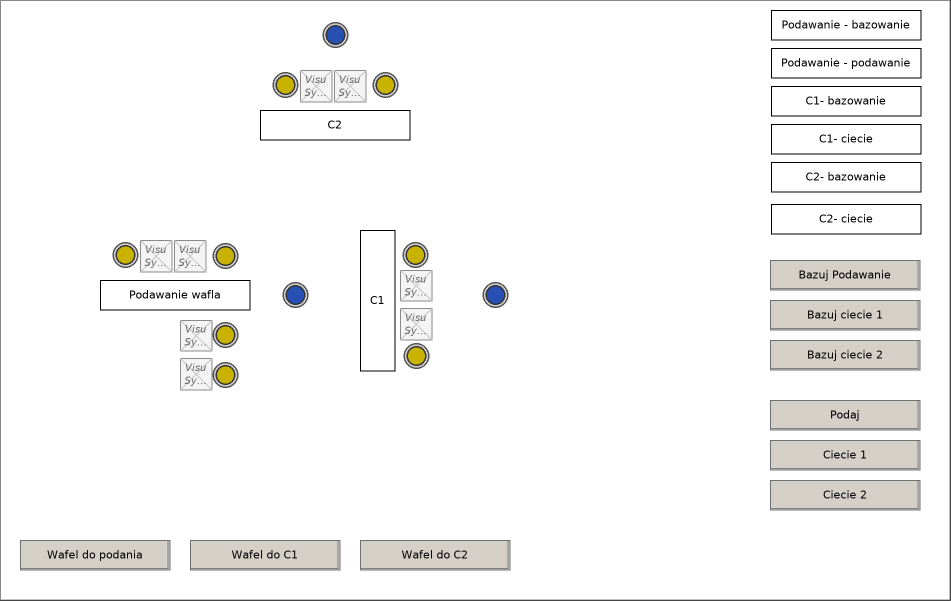
VISUALIZATION Symulacja  // 951x601
VAR_IN_OUT
	stDane									: DUT_Wizualizacja_SymulacjaDane;
END_VAR
    Line (950,0) (950,600)
    Line (0,600) (950,600)
    Rectangle (100,280 150x30), "Podawanie wafla"
    Rectangle (360,230 35x141), "C1"
    Rectangle (260,110 150x30), "C2"
    Lamp1 (401,341 31x30), variable: stDane.bCiecie1_Poczatek, style: Lamp-Lamp1-Yellow
    Lamp1 (400,240 31x30), variable: stDane.bCiecie1_Koniec, style: Lamp-Lamp1-Yellow
    Lamp1 (270,70 31x30), variable: stDane.bCiecie2_Poczatek, style: Lamp-Lamp1-Yellow
    Lamp1 (370,70 31x30), variable: stDane.bCiecie2_Koniec, style: Lamp-Lamp1-Yellow
    Lamp1 (110,240 31x30), variable: stDane.bPodawaniePrzesuwanieKoniec, style: Lamp-Lamp1-Yellow
    Lamp1 (210,241 31x30), variable: stDane.bPodawaniePrzesuwaniePoczatek, style: Lamp-Lamp1-Yellow
    Lamp1 (210,320 31x30), variable: stDane.bPodawanieZabierakKoniec, style: Lamp-Lamp1-Yellow
    Lamp1 (210,360 31x30), variable: stDane.bPodawanieZabierakPoczatek, style: Lamp-Lamp1-Yellow
    Lamp1 (280,280 31x30), variable: stDane.bCzujnikWaflaDoPodania, style: Lamp-Lamp1-Blue
    Lamp1 (480,280 31x30), variable: stDane.bCzujnikWaflaDoCiecia1, style: Lamp-Lamp1-Blue
    Lamp1 (320,20 31x30), variable: stDane.bCzujnikWaflaDoCiecia2, style: Lamp-Lamp1-Blue
    Rectangle (771,10 150x30), "Podawanie - bazowanie", colour toggle: stDane.stStanySilownikow.bPodawanie_Bazowanie
    Rectangle (771,48 150x30), "Podawanie - podawanie", colour toggle: stDane.stStanySilownikow.bPodawanie_Podawanie
    Rectangle (771,86 150x30), "C1- bazowanie", colour toggle: stDane.stStanySilownikow.bCiecie1_Bazowanie
    Rectangle (771,124 150x30), "C1- ciecie", colour toggle: stDane.stStanySilownikow.bCiecie1_Ciecie
    Rectangle (771,162 150x30), "C2- bazowanie", colour toggle: stDane.stStanySilownikow.bCiecie2_Bazowanie
    Rectangle (771,204 150x30), "C2- ciecie", colour toggle: stDane.stStanySilownikow.bCiecie2_Ciecie
    Image (180,358 32x32), invisible if: Not stDane.stStanySilownikow.bPodawanie_Zabierak_WStronePoczatku, image: VisuSymbols.Symbols.ArrowBoldDown
    Image (180,320 32x31), invisible if: Not stDane.stStanySilownikow.bPodawanie_zabierak_WStroneKonca, image: VisuSymbols.Symbols.ArrowBoldUp
    Image (140,240 32x32), invisible if: Not stDane.stStanySilownikow.bPodawanie_Przesuwanie_WStroneKonca, image: VisuSymbols.Symbols.ArrowBoldLeft
    Image (174,240 32x32), invisible if: Not stDane.stStanySilownikow.bPodawanie_Przesuwanie_WStronePoczatku, image: VisuSymbols.Symbols.ArrowBoldRight
    Image (400,308 32x32), invisible if: Not stDane.stStanySilownikow.bCiecie1_Naped_WStronePoczatku, image: VisuSymbols.Symbols.ArrowBoldDown
    Image (400,270 32x31), invisible if: Not stDane.stStanySilownikow.bCiecie1_Naped_WStroneKonca, image: VisuSymbols.Symbols.ArrowBoldUp
    Image (300,70 32x32), invisible if: Not stDane.stStanySilownikow.bCiecie2_Naped_WStronePoczatku, image: VisuSymbols.Symbols.ArrowBoldLeft
    Image (334,70 32x32), invisible if: Not stDane.stStanySilownikow.bCiecie2_Naped_WStroneKonca, image: VisuSymbols.Symbols.ArrowBoldRight
    Button (770,260 150x30), "Bazuj Podawanie", invisible if: stDane.eTrybPracy <> E_PMLUnitMode.SEMIAUTOMATIC
        tap stDane.bPodawanieBazuj
    Button (770,300 150x30), "Bazuj ciecie 1", invisible if: stDane.eTrybPracy <> E_PMLUnitMode.SEMIAUTOMATIC
        tap stDane.bCiecie1Bazuj
    Button (770,340 150x30), "Bazuj ciecie 2", invisible if: stDane.eTrybPracy <> E_PMLUnitMode.SEMIAUTOMATIC
        tap stDane.bCiecie2Bazuj
    Button (770,400 150x30), "Podaj", invisible if: stDane.eTrybPracy <> E_PMLUnitMode.SEMIAUTOMATIC
        tap stDane.bPodawaniePodaj
    Button (770,440 150x30), "Ciecie 1", invisible if: stDane.eTrybPracy <> E_PMLUnitMode.SEMIAUTOMATIC
        tap stDane.bCiecie1Tnij
    Button (770,480 150x30), "Ciecie 2", invisible if: stDane.eTrybPracy <> E_PMLUnitMode.SEMIAUTOMATIC
        tap stDane.bCiecie2Tnij
    Button (20,540 150x30), "Wafel do podania", invisible if: stDane.eTrybPracy <> E_PMLUnitMode.SEMIAUTOMATIC
        toggle stDane.bCzujnikWaflaDoPodania
    Button (190,540 150x30), "Wafel do C1", invisible if: stDane.eTrybPracy <> E_PMLUnitMode.SEMIAUTOMATIC
        toggle stDane.bCzujnikWaflaDoCiecia1
    Button (360,540 150x30), "Wafel do C2", invisible if: stDane.eTrybPracy <> E_PMLUnitMode.SEMIAUTOMATIC
        toggle stDane.bCzujnikWaflaDoCiecia2
END_VISUALIZATION

(* stored: Version 1.1.0.1, ProductVersion 3.1.4024.11
   Visu Symulacja: Id {a07c3a47-53ac-43b1-9a89-64147dd50306} *)
